(* Logix 5000 project; controller ECE4350_Lab8_AngelinoLefevers 5069-L306ERM rev 30.11; software revision 30.00 *)

TASK MainTask (continuous, watchdog 500 ms) : MainProgram

MODULES
   Local : 5069-L306ERM (5069 0, rev 30.11)
      Digital_IN : 5069-IB16 (5069 1, rev 2.1, StandardDataDriven RPI 5 ms)
      Analog_IN : vendor 1 type 115 code 314 (5069 2, rev 2.1, StandardDataDriven RPI 100 ms)
      Analog_OUT : vendor 1 type 115 code 320 (5069 4, rev 2.1, StandardDataDriven RPI 80 ms)
      Digital_OUT : 5069-OB16 (5069 3, rev 2.1, StandardDataDriven RPI 5 ms)
END_MODULES

PROGRAM MainProgram   (* main routine MainRoutine *)
VAR
   Degrees : REAL;
   GreenButton : ALIAS FOR Local:1:I.Pt01.Data;   // Normally Open
   GreenLight : ALIAS FOR Local:3:O.Pt01.Data;
   Inputted_Value : REAL;
   LB : BOOL;
   MOT_NUM : BOOL;
   MOT_POT : BOOL;
   Motor : ALIAS FOR Local:4:O.Ch00.Data;
   Outside_Range : BOOL;
   POT_Value : REAL;
   Potentiometer : ALIAS FOR Local:2:I.Ch00.Data;
   PT : BOOL;   // Potentiometer Toggle
   R1 : BOOL;
   R2 : BOOL;
   R3 : BOOL;
   R4 : BOOL;
   R5 : BOOL;
   RedButton : ALIAS FOR Local:1:I.Pt00.Data;   // Normally Closed
   RedLight : ALIAS FOR Local:3:O.Pt00.Data;
   Relay_1 : ALIAS FOR Local:3:O.Pt02.Data;
   Relay_2 : ALIAS FOR Local:3:O.Pt03.Data;
   Relay_3 : ALIAS FOR Local:3:O.Pt04.Data;
   Relay_4 : ALIAS FOR Local:3:O.Pt05.Data;
   Relay_5 : ALIAS FOR Local:3:O.Pt06.Data;
   Thermistor : ALIAS FOR Local:2:I.Ch01.Data;
   TM1 : TIMER := (PRE := 20000);
   ToggleLeft : ALIAS FOR Local:1:I.Pt03.Data;
   ToggleRight : ALIAS FOR Local:1:I.Pt02.Data;
END_VAR

ROUTINE MainRoutine   (* ladder *)
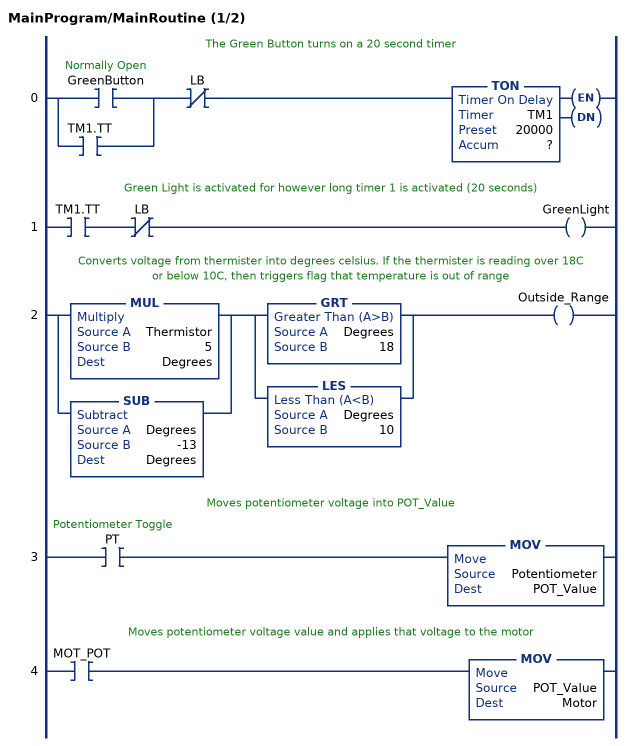
   // The Green Button turns on a 20 second timer
   0: [XIC(GreenButton) ,XIC(TM1.TT) ]XIO(LB)TON(TM1,?,?);
   // Green Light is activated for however long timer 1 is activated (20 seconds)
   1: XIC(TM1.TT)XIO(LB)OTE(GreenLight);
   // Converts voltage from thermister into degrees celsius. If the thermister is reading over 18C or below 10C, then triggers flag that temperature is out of range
   2: [MUL(Thermistor,5,Degrees) ,SUB(Degrees,-13,Degrees) ][GRT(Degrees,18) ,LES(Degrees,10) ]OTE(Outside_Range);
   // Moves potentiometer voltage into POT_Value
   3: XIC(PT)MOV(Potentiometer,POT_Value);
   // Moves potentiometer voltage value and applies that voltage to the motor
   4: XIC(MOT_POT)MOV(POT_Value,Motor);
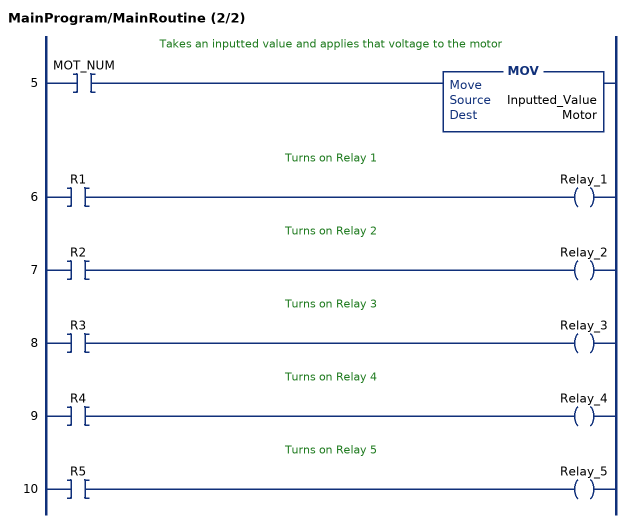
   // Takes an inputted value and applies that voltage to the motor
   5: XIC(MOT_NUM)MOV(Inputted_Value,Motor);
   // Turns on Relay 1
   6: XIC(R1)OTE(Relay_1);
   // Turns on Relay 2
   7: XIC(R2)OTE(Relay_2);
   // Turns on Relay 3
   8: XIC(R3)OTE(Relay_3);
   // Turns on Relay 4
   9: XIC(R4)OTE(Relay_4);
   // Turns on Relay 5
   10: XIC(R5)OTE(Relay_5);
END_ROUTINE
END_PROGRAM
